FUNCTION_BLOCK CLIENT_0_21 (* 4-Input,4-Output Client Interface *)
  (* Standard: 61499-1; Classification: Communications *)
  (* Version 0.0, 2001-05-23, JHC, Rockwell Automation *)
  (* Compiler header: package fb.rt.net; *)
  (* Compiler Java IBM VisualAge 3.0 *)
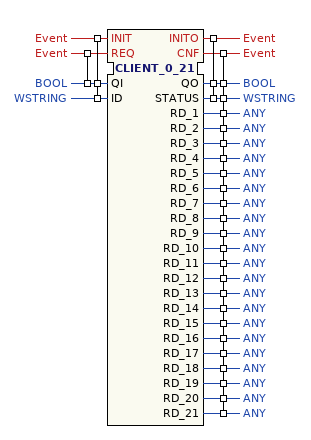
  EVENT_INPUT
    INIT WITH QI, ID; (* Service Initialization *)
    REQ WITH QI; (* Service Request *)
  END_EVENT
  EVENT_OUTPUT
    INITO WITH QO, STATUS; (* Initialization Confirm *)
    CNF WITH QO, STATUS, RD_1, RD_2, RD_3, RD_4, RD_5, RD_6, RD_7, RD_8, RD_9, RD_10, RD_11, RD_12, RD_13, RD_14, RD_15, RD_16, RD_17, RD_18, RD_19, RD_20, RD_21; (* Service Confirmation *)
  END_EVENT
  VAR_INPUT
    QI : BOOL; (* Event Input Qualifier *)
    ID : WSTRING; (* Connection Identifier *)
  END_VAR
  VAR_OUTPUT
    QO : BOOL; (* Event Output Qualifier *)
    STATUS : WSTRING; (* Service Status *)
    RD_1 : ANY; (* Received Data *)
    RD_2 : ANY; (* Received Data *)
    RD_3 : ANY; (* Received Data *)
    RD_4 : ANY; (* Received Data *)
    RD_5 : ANY; (* Received Data *)
    RD_6 : ANY; (* Received Data *)
    RD_7 : ANY; (* Received Data *)
    RD_8 : ANY; (* Received Data *)
    RD_9 : ANY; (* Received Data *)
    RD_10 : ANY; (* Received Data *)
    RD_11 : ANY; (* Received Data *)
    RD_12 : ANY; (* Received Data *)
    RD_13 : ANY; (* Received Data *)
    RD_14 : ANY; (* Received Data *)
    RD_15 : ANY; (* Received Data *)
    RD_16 : ANY; (* Received Data *)
    RD_17 : ANY; (* Received Data *)
    RD_18 : ANY; (* Received Data *)
    RD_19 : ANY; (* Received Data *)
    RD_20 : ANY; (* Received Data *)
    RD_21 : ANY; (* Received Data *)
  END_VAR
END_FUNCTION_BLOCK
